RoboDK station: Tutorial Station.rdk

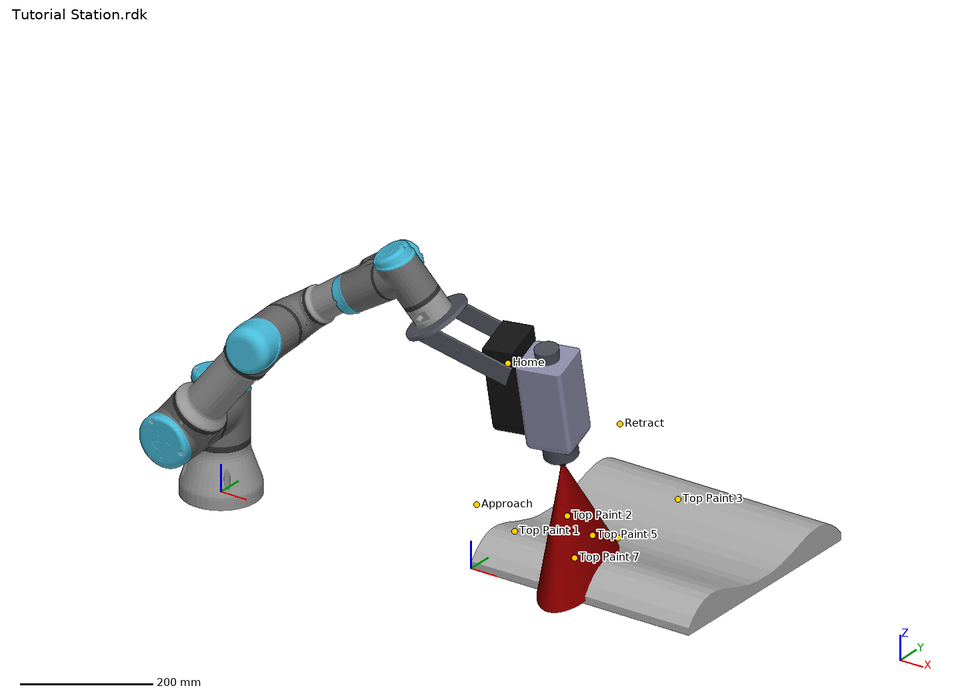
[picture v0: the station drawn from its stored meshes, robots at their saved joint values, targets as dots, program paths as lines]
Station Tutorial Station (saved by RoboDK 5.8.0). Poses are relative to the parent item; angles as X-Y-Z fixed-axis rotations.
Station parameters (name, value as stored): LIN64
  - frame UR3 Base at (0, 0, 0) mm
    - robot UR3: 6 axes, payload 3 kg, reach 500 mm, repeatability 0.1 mm, weight 11 kg
        modified DH rows (alpha deg, a mm, theta deg, d mm): 0, 0, 0, 151.9; 90, 0, 180, 0; 0, 243.65, 0, 0; 0, 213, 0, 110.4; -90, 0, 0, 83.4; 90, 0, 180, 82.4
        joint limits [-360, -360, -360, -360, -360, -360] to [360, 360, 360, 360, 360, 360]; home [0, -90, -90, 0, 90, 0]; saved at [3.337, -127.931, -15.921, -94.792, 102.869, 90.751]
      - tool Paint gun, TCP at (50, 0, 450) mm, rotated rx 0 ry 30 rz 0 deg, size 203.2 x 279.7 x 471.5 mm
  - frame Frame 2 at (460.12, 0, 0) mm
    - object Object Inspection at (0, 0, 0) mm, size 400 x 400 x 46.2 mm, geometry from Object Inspection.stl
    - target Home (Cartesian target) at (145.4, -110.4, 428.95) mm, rotated rx -180 ry 60 rz -180 deg; joints [0, -90, -90, 0, 90, 90] of UR3
    - target Approach (Cartesian target) at (9.63, 1.78, 108.65) mm, rotated rx -180 ry -2.15 rz -166.19 deg; joints [13.81, -103.499, -21.273, -117.377, 90, 90] of UR3
    - target Retract (Cartesian target) at (15.32, 370.14, 99.2) mm, rotated rx 179.62 ry 7.58 rz -164.97 deg; joints [217.468, -65.591, 28.198, -88.14, -103.15, 108.283] of UR3
    - target Top Paint 1 (Cartesian target) at (35, 64.68, 45.84) mm, rotated rx -178.05 ry 0.03 rz -180 deg; joints [173.735, -90.4, 64.146, -93.797, -88.548, 83.603] of UR3
    - target Top Paint 2 (Cartesian target) at (34.99, 203.51, 16.09) mm, rotated rx 171.91 ry -0.45 rz -179.97 deg; joints [185.006, -87.45, 70.598, -103.383, -85.492, 98.393] of UR3
    - target Top Paint 3 (Cartesian target) at (166.34, 305.56, 40.5) mm, rotated rx 164.25 ry 8.39 rz -152.64 deg; joints [22.092, -155.651, 27.204, -103.322, 106.9, 93.769] of UR3
    - target Top Paint 5 (Cartesian target) at (108.72, 164.13, 20.72) mm, rotated rx -172.09 ry 0.43 rz -179.97 deg; joints [49.508, -138.487, 9.12, -125.033, 62.46, 133.539] of UR3
    - target Top Paint 6 (Cartesian target) at (143.08, 182.35, 18.47) mm, rotated rx -179.51 ry -0.08 rz -170.52 deg; joints [36.906, -126.963, -18.568, -97.589, 76.335, 114.012] of UR3
    - target Top Paint 7 (Cartesian target) at (158.61, 44.91, 44) mm, rotated rx 168.63 ry 1.84 rz -170.9 deg; joints [3.337, -127.931, -15.921, -94.792, 102.869, 90.751] of UR3
